{attribute 'GeneratedUsingTerminal: EL3423-0000-0016'}
{attribute addProperty BoxType "EL3423-0000-0016"}
{attribute addProperty Id "Apparent_EnergyAT %I*LINT8Apparent_Positive_EnergyAT %I*ULINT8Apparent_Negative_EnergyAT %I*ULINT8"}
{attribute addProperty CRC "2408839557"}
{attribute addProperty Size "24"}
TYPE Total_Apparent_8F93F985 EXTENDS InputBase_8311D824 :
STRUCT
	{attribute addProperty Name "Apparent_Energy"}
	Apparent_Energy AT %I* : LINT;
	{attribute addProperty Name "Apparent_Positive_Energy"}
	Apparent_Positive_Energy AT %I* : ULINT;
	{attribute addProperty Name "Apparent_Negative_Energy"}
	Apparent_Negative_Energy AT %I* : ULINT;
END_STRUCT
END_TYPE

(* stored: Version 1.2.0.0, ProductVersion 3.1.4024.11
   DUT Total_Apparent_8F93F985: Id {244da7ce-c718-4be5-87cc-bc6836e61c94} *)
